// TIA Portal project "Gip & module 1" (V14)

(* hardware
DEVICE "S7-1200 station_1"  S7-1200 Station
   slot 0: "Rack_0"  S7-1200 Rack  Rack  V1.0
   slot 1: "PLC_1"  CPU 1214C DC/DC/DC  6ES7 214-1AG31-0XB0  V3.0
      slot 3: "AQ 1x12BIT_1"  AQ1 signal board  6ES7 232-4HA30-0XB0  V1.0
   slot 101: "CM 1243-5"  CM 1243-5  6GK7 243-5DX30-0XE0  V1.3
DEVICE "HMI_1"  KTP700 Basic PN
   slot 0: "KTP700 Basic PN"  KTP700 Basic PN  6AV2 123-2GB03-0AX0  14.0.1.0
   slot 1: "HMI_RT_1"  KTP700 Basic PN  6AV2 123-2GB03-0AX0  14.0.1.0
   slot 5: "HMI_1.IE_CP_1"  PROFINET Interface  14.0.1.0
      slot 1: "PROFINET Interface_1"  PROFINET Interface
         slot 1: "Port_1"  Port
DEVICE "GSD device_1"  GSD.Device
   slot 0: "Rack_0"  Rail
*)

// ===== PLC "PLC_1"  CPU 1214C DC/DC/DC =====

VAR_GLOBAL   // PLC tag table "Default tag table"
   "sensor" AT %I0.0 : Bool;
   "TBG_B_Achter" AT %I2.0 : Bool;
   "TBG_B_Midden" AT %I2.1 : Bool;
   "TBG_B_Voor" AT %I2.2 : Bool;
   "TBK_B_Achter" AT %I2.3 : Bool;
   "TBK_B_Midden" AT %I2.4 : Bool;
   "TBK_B_Voor" AT %I2.5 : Bool;
   "Brug_B_G" AT %I2.6 : Bool;
   "Brug_B_K" AT %I2.7 : Bool;
   "Brug_B_A" AT %I3.0 : Bool;
   "K1_B_Boven" AT %I3.1 : Bool;
   "K1_B_Beneden" AT %I3.2 : Bool;
   "K1_B_Vacium" AT %I3.3 : Bool;
   "Druk" AT %I3.5 : Bool;
   "TBA_B" AT %I3.4 : Bool;
   "TBG_M_Achter" AT %Q2.0 : Bool;
   "TBG_M_Voor" AT %Q2.1 : Bool;
   "TBK_M_Achter" AT %Q2.2 : Bool;
   "TBK_M_Voor" AT %Q2.3 : Bool;
   "TBA_M_Achter" AT %Q2.4 : Bool;
   "TBA_M_Voor" AT %Q2.5 : Bool;
   "Brug_M_Links" AT %Q2.6 : Bool;
   "Brug_M_Rechts" AT %Q2.7 : Bool;
   "K1_Boven" AT %Q3.0 : Bool;
   "K1_Beneden" AT %Q3.1 : Bool;
   "K1_Vacium" AT %Q3.2 : Bool;
   "Veilig opstartventiel" AT %Q3.3 : Bool;
   "New_Order" AT %M0.1 : Bool;
   "TBG_M_Achter_SR" AT %M10.0 : Bool;
   "TBG_M_Voor_SR" AT %M10.1 : Bool;
   "TBK_M_Achter_SR" AT %M10.2 : Bool;
   "TBK_M_Voor_SR" AT %M10.3 : Bool;
   "TBA_M_Achter_SR" AT %M10.4 : Bool;
   "TBA_M_Voor_SR" AT %M10.5 : Bool;
   "Brug_M_Rechts_SR" AT %M10.6 : Bool;
   "Brug_M_Links_SR" AT %M10.7 : Bool;
   "K1_Boven_SR" AT %M11.0 : Bool;
   "K1_Beneden_SR" AT %M11.1 : Bool;
   "K1_Vacium_SR" AT %M11.2 : Bool;
   "Reset_SR" AT %M11.3 : Bool;
   "S/S_SR" AT %M11.4 : Bool;
   "Start" AT %M20.0 : Bool;
   "Stop" AT %M20.1 : Bool;
   "Reset" AT %M20.2 : Bool;
   "Klein" AT %M20.3 : Bool;
   "Groot" AT %M20.4 : Bool;
   "Reset_Hmi" AT %M20.5 : Bool;
   "Test" AT %M20.6 : Bool;
   "Test_SR" AT %M11.5 : Bool;
   "Stop Alles" AT %M20.7 : Bool;
   "Proces_Order" AT %M21.0 : Bool;
END_VAR

DATA_BLOCK "Data_block_1"   // DB100
{ S7_Optimized_Access := 'FALSE' }
VERSION : 0.1
   VAR
      R : Int := 0;
      G : Int := 0;
      "B" : Int := 0;
      "G/K" : Int := 0;
      Locatie : Int;
      New : Bool := False;
   END_VAR
BEGIN
END_DATA_BLOCK

// folder: System blocks/Program resources

DATA_BLOCK "IEC_Timer_0_DB"   // DB1
{ S7_Optimized_Access := 'TRUE' }
AUTHOR : Simatic
FAMILY : IEC
NAME : IEC_TMR
VERSION : 1.0
// stored: InstanceOfName IEC_TIMER
"IEC_TIMER"
BEGIN
END_DATA_BLOCK

// folder: (top level)

FUNCTION "Block_1" : Void   // FC1, SCL
{ S7_Optimized_Access := 'TRUE' }
VERSION : 0.1
BEGIN
   IF "New_Order" = TRUE THEN
       "Data_block_1".New := TRUE;
       "New_Order" := FALSE;
   END_IF;

   IF "Data_block_1"."G/K" = 1 THEN
       "Groot" := TRUE;
       "Klein" := FALSE;
   END_IF;

   IF "Data_block_1"."G/K" = 0 THEN
       "Groot" := FALSE;
       "Klein" := TRUE;
   END_IF;
END_FUNCTION

FUNCTION "S/S + Reset + Druk" : Void   // FC2, LAD
{ S7_Optimized_Access := 'TRUE' }
VERSION : 0.1
BEGIN

REGION Network 1: S+R/S veilig opstartvetiel
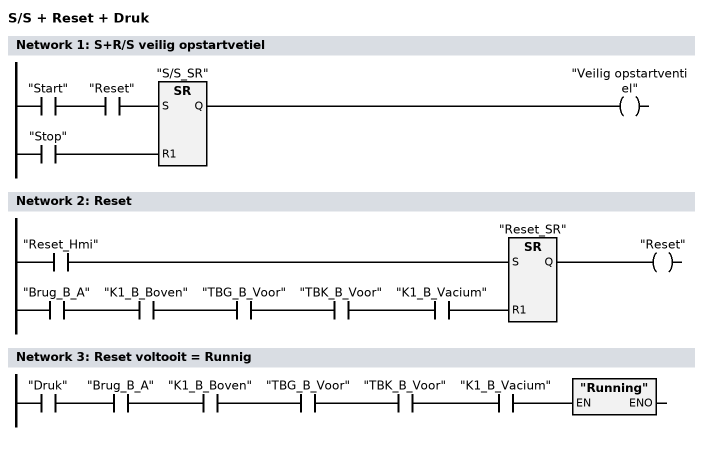
   RUNG wire#powerrail
      Contact( "Start" )
      Contact( "Reset" )
      S_SR(operand := "S/S_SR", r1 := wire#w1)
      Coil( "Veilig opstartventiel" )
   END_RUNG
   RUNG wire#powerrail
      Contact( "Stop" )
   END_RUNG wire#w1
   // the same network as SCL:
   IF "Start" AND "Reset" THEN
       "S/S_SR" := TRUE;   // SR flip-flop
   END_IF;
   IF "Stop" THEN "S/S_SR" := FALSE; END_IF;
   "Veilig opstartventiel" := "S/S_SR";
END_REGION

REGION Network 2: Reset
   RUNG wire#powerrail
      Contact( "Reset_Hmi" )
      S_SR(operand := "Reset_SR", r1 := wire#w1)
      Coil( "Reset" )
   END_RUNG
   RUNG wire#powerrail
      Contact( "Brug_B_A" )
      Contact( "K1_B_Boven" )
      Contact( "TBG_B_Voor" )
      Contact( "TBK_B_Voor" )
      Contact( "K1_B_Vacium" )
   END_RUNG wire#w1
   // the same network as SCL:
   IF "Reset_Hmi" THEN
       "Reset_SR" := TRUE;   // SR flip-flop
   END_IF;
   IF "Brug_B_A" AND "K1_B_Boven" AND "TBG_B_Voor" AND "TBK_B_Voor" AND "K1_B_Vacium" THEN
       "Reset_SR" := FALSE;
   END_IF;
   "Reset" := "Reset_SR";
END_REGION

REGION Network 3: Reset voltooit = Runnig
   RUNG wire#powerrail
      Contact( "Druk" )
      Contact( "Brug_B_A" )
      Contact( "K1_B_Boven" )
      Contact( "TBG_B_Voor" )
      Contact( "TBK_B_Voor" )
      Contact( "K1_B_Vacium" )
      "Running"()
   END_RUNG
   // the same network as SCL:
   IF "Druk" AND "Brug_B_A" AND "K1_B_Boven" AND "TBG_B_Voor" AND "TBK_B_Voor" AND "K1_B_Vacium" THEN
       "Running"();
   END_IF;
END_REGION
END_FUNCTION

FUNCTION "Running" : Void   // FC3, LAD
{ S7_Optimized_Access := 'TRUE' }
VERSION : 0.1
BEGIN

REGION Network 1: Grote bakjes naar achter
END_REGION

REGION Network 2: Grote bakjes naar voor
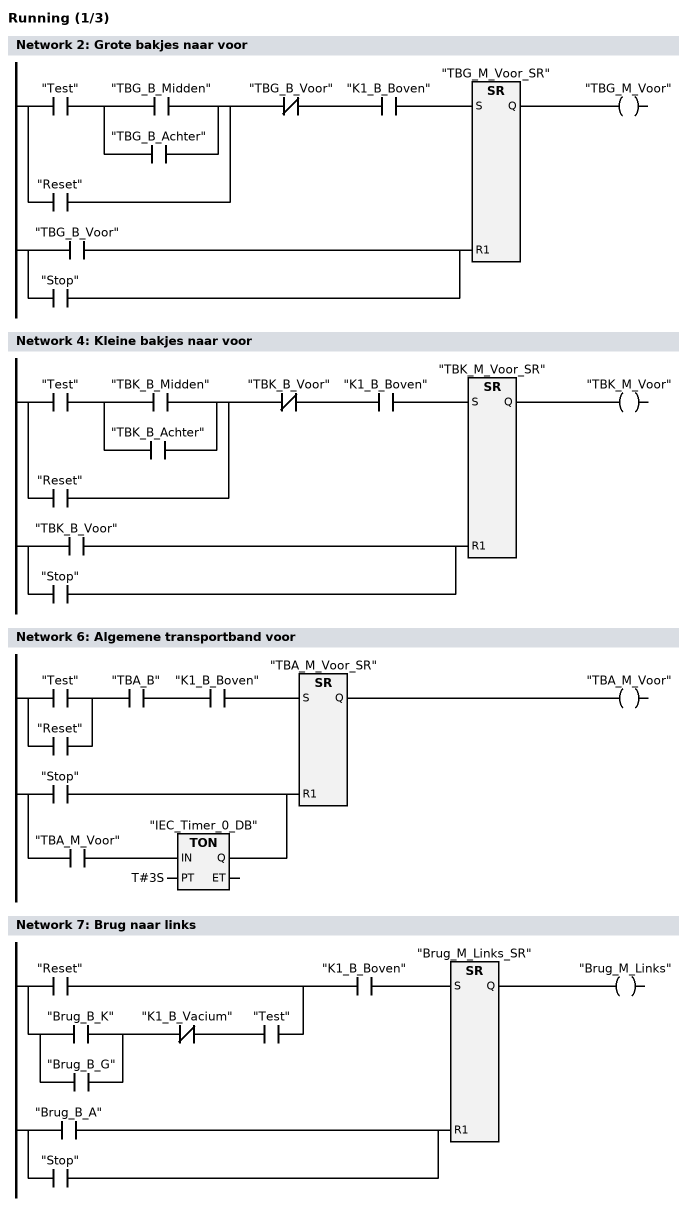
   RUNG wire#powerrail
      Contact( "Test" )
      wire#w1
      Contact( "TBG_B_Midden" )
      wire#w2
      I_Contact( "TBG_B_Voor" )
      Contact( "K1_B_Boven" )
      S_SR(operand := "TBG_M_Voor_SR", r1 := wire#w3)
      Coil( "TBG_M_Voor" )
   END_RUNG
   RUNG wire#w1
      Contact( "TBG_B_Achter" )
   END_RUNG wire#w2
   RUNG wire#powerrail
      Contact( "Reset" )
   END_RUNG wire#w2
   RUNG wire#powerrail
      Contact( "TBG_B_Voor" )
   END_RUNG wire#w3
   RUNG wire#powerrail
      Contact( "Stop" )
   END_RUNG wire#w3
   // the same network as SCL:
   IF (("Test" AND ("TBG_B_Midden" OR "TBG_B_Achter")) OR "Reset") AND NOT "TBG_B_Voor" AND "K1_B_Boven" THEN
       "TBG_M_Voor_SR" := TRUE;   // SR flip-flop
   END_IF;
   IF "TBG_B_Voor" OR "Stop" THEN "TBG_M_Voor_SR" := FALSE; END_IF;
   "TBG_M_Voor" := "TBG_M_Voor_SR";
END_REGION

REGION Network 3: Kleine bakjes naar achter
END_REGION

REGION Network 4: Kleine bakjes naar voor
   RUNG wire#powerrail
      Contact( "Test" )
      wire#w1
      Contact( "TBK_B_Midden" )
      wire#w2
      I_Contact( "TBK_B_Voor" )
      Contact( "K1_B_Boven" )
      S_SR(operand := "TBK_M_Voor_SR", r1 := wire#w3)
      Coil( "TBK_M_Voor" )
   END_RUNG
   RUNG wire#w1
      Contact( "TBK_B_Achter" )
   END_RUNG wire#w2
   RUNG wire#powerrail
      Contact( "Reset" )
   END_RUNG wire#w2
   RUNG wire#powerrail
      Contact( "TBK_B_Voor" )
   END_RUNG wire#w3
   RUNG wire#powerrail
      Contact( "Stop" )
   END_RUNG wire#w3
   // the same network as SCL:
   IF (("Test" AND ("TBK_B_Midden" OR "TBK_B_Achter")) OR "Reset") AND NOT "TBK_B_Voor" AND "K1_B_Boven" THEN
       "TBK_M_Voor_SR" := TRUE;   // SR flip-flop
   END_IF;
   IF "TBK_B_Voor" OR "Stop" THEN "TBK_M_Voor_SR" := FALSE; END_IF;
   "TBK_M_Voor" := "TBK_M_Voor_SR";
END_REGION

REGION Network 5: Algemene transportband achter
END_REGION

REGION Network 6: Algemene transportband voor
   "IEC_Timer_0_DB".TON(IN := "TBA_M_Voor", PT := T#3S);
   IF ("Test" OR "Reset") AND "TBA_B" AND "K1_B_Boven" THEN
       "TBA_M_Voor_SR" := TRUE;   // SR flip-flop
   END_IF;
   IF "Stop" OR "IEC_Timer_0_DB".Q THEN "TBA_M_Voor_SR" := FALSE; END_IF;
   "TBA_M_Voor" := "TBA_M_Voor_SR";
END_REGION

REGION Network 7: Brug naar links
   RUNG wire#powerrail
      Contact( "Reset" )
      wire#w1
      Contact( "K1_B_Boven" )
      S_SR(operand := "Brug_M_Links_SR", r1 := wire#w3)
      Coil( "Brug_M_Links" )
   END_RUNG
   RUNG wire#powerrail
      Contact( "Brug_B_K" )
      wire#w2
      I_Contact( "K1_B_Vacium" )
      Contact( "Test" )
   END_RUNG wire#w1
   RUNG wire#powerrail
      Contact( "Brug_B_G" )
   END_RUNG wire#w2
   RUNG wire#powerrail
      Contact( "Brug_B_A" )
   END_RUNG wire#w3
   RUNG wire#powerrail
      Contact( "Stop" )
   END_RUNG wire#w3
   // the same network as SCL:
   IF ("Reset" OR (("Brug_B_K" OR "Brug_B_G") AND NOT "K1_B_Vacium" AND "Test")) AND "K1_B_Boven" THEN
       "Brug_M_Links_SR" := TRUE;   // SR flip-flop
   END_IF;
   IF "Brug_B_A" OR "Stop" THEN "Brug_M_Links_SR" := FALSE; END_IF;
   "Brug_M_Links" := "Brug_M_Links_SR";
END_REGION

REGION Network 8: Brug naar rechts
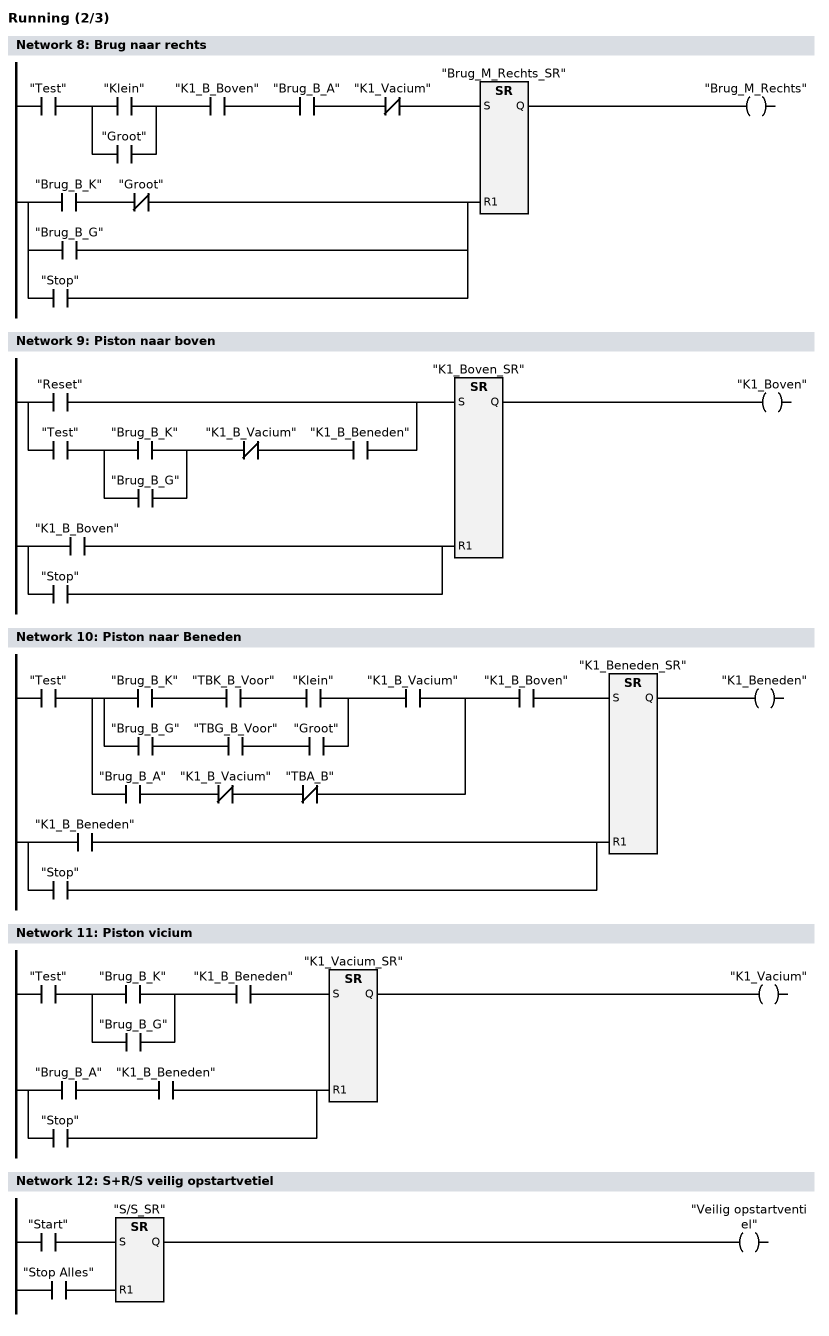
   RUNG wire#powerrail
      Contact( "Test" )
      wire#w1
      Contact( "Klein" )
      wire#w2
      Contact( "K1_B_Boven" )
      Contact( "Brug_B_A" )
      I_Contact( "K1_Vacium" )
      S_SR(operand := "Brug_M_Rechts_SR", r1 := wire#w3)
      Coil( "Brug_M_Rechts" )
   END_RUNG
   RUNG wire#w1
      Contact( "Groot" )
   END_RUNG wire#w2
   RUNG wire#powerrail
      Contact( "Brug_B_K" )
      I_Contact( "Groot" )
   END_RUNG wire#w3
   RUNG wire#powerrail
      Contact( "Brug_B_G" )
   END_RUNG wire#w3
   RUNG wire#powerrail
      Contact( "Stop" )
   END_RUNG wire#w3
   // the same network as SCL:
   IF "Test" AND ("Klein" OR "Groot") AND "K1_B_Boven" AND "Brug_B_A" AND NOT "K1_Vacium" THEN
       "Brug_M_Rechts_SR" := TRUE;   // SR flip-flop
   END_IF;
   IF ("Brug_B_K" AND NOT "Groot") OR "Brug_B_G" OR "Stop" THEN "Brug_M_Rechts_SR" := FALSE; END_IF;
   "Brug_M_Rechts" := "Brug_M_Rechts_SR";
END_REGION

REGION Network 9: Piston naar boven
   RUNG wire#powerrail
      Contact( "Reset" )
      wire#w1
      S_SR(operand := "K1_Boven_SR", r1 := wire#w4)
      Coil( "K1_Boven" )
   END_RUNG
   RUNG wire#powerrail
      Contact( "Test" )
      wire#w2
      Contact( "Brug_B_K" )
      wire#w3
      I_Contact( "K1_B_Vacium" )
      Contact( "K1_B_Beneden" )
   END_RUNG wire#w1
   RUNG wire#w2
      Contact( "Brug_B_G" )
   END_RUNG wire#w3
   RUNG wire#powerrail
      Contact( "K1_B_Boven" )
   END_RUNG wire#w4
   RUNG wire#powerrail
      Contact( "Stop" )
   END_RUNG wire#w4
   // the same network as SCL:
   IF "Reset" OR ("Test" AND ("Brug_B_K" OR "Brug_B_G") AND NOT "K1_B_Vacium" AND "K1_B_Beneden") THEN
       "K1_Boven_SR" := TRUE;   // SR flip-flop
   END_IF;
   IF "K1_B_Boven" OR "Stop" THEN "K1_Boven_SR" := FALSE; END_IF;
   "K1_Boven" := "K1_Boven_SR";
END_REGION

REGION Network 10: Piston naar Beneden
   RUNG wire#powerrail
      Contact( "Test" )
      wire#w1
      Contact( "Brug_B_K" )
      Contact( "TBK_B_Voor" )
      Contact( "Klein" )
      wire#w2
      Contact( "K1_B_Vacium" )
      wire#w3
      Contact( "K1_B_Boven" )
      S_SR(operand := "K1_Beneden_SR", r1 := wire#w4)
      Coil( "K1_Beneden" )
   END_RUNG
   RUNG wire#w1
      Contact( "Brug_B_G" )
      Contact( "TBG_B_Voor" )
      Contact( "Groot" )
   END_RUNG wire#w2
   RUNG wire#w1
      Contact( "Brug_B_A" )
      I_Contact( "K1_B_Vacium" )
      I_Contact( "TBA_B" )
   END_RUNG wire#w3
   RUNG wire#powerrail
      Contact( "K1_B_Beneden" )
   END_RUNG wire#w4
   RUNG wire#powerrail
      Contact( "Stop" )
   END_RUNG wire#w4
   // the same network as SCL:
   IF "Test" AND (((("Brug_B_K" AND "TBK_B_Voor" AND "Klein") OR ("Brug_B_G" AND "TBG_B_Voor" AND "Groot")) AND "K1_B_Vacium") OR ("Brug_B_A" AND NOT "K1_B_Vacium" AND NOT "TBA_B")) AND "K1_B_Boven" THEN
       "K1_Beneden_SR" := TRUE;   // SR flip-flop
   END_IF;
   IF "K1_B_Beneden" OR "Stop" THEN "K1_Beneden_SR" := FALSE; END_IF;
   "K1_Beneden" := "K1_Beneden_SR";
END_REGION

REGION Network 11: Piston vicium
   RUNG wire#powerrail
      Contact( "Test" )
      wire#w1
      Contact( "Brug_B_K" )
      wire#w2
      Contact( "K1_B_Beneden" )
      S_SR(operand := "K1_Vacium_SR", r1 := wire#w3)
      Coil( "K1_Vacium" )
   END_RUNG
   RUNG wire#w1
      Contact( "Brug_B_G" )
   END_RUNG wire#w2
   RUNG wire#powerrail
      Contact( "Brug_B_A" )
      Contact( "K1_B_Beneden" )
   END_RUNG wire#w3
   RUNG wire#powerrail
      Contact( "Stop" )
   END_RUNG wire#w3
   // the same network as SCL:
   IF "Test" AND ("Brug_B_K" OR "Brug_B_G") AND "K1_B_Beneden" THEN
       "K1_Vacium_SR" := TRUE;   // SR flip-flop
   END_IF;
   IF ("Brug_B_A" AND "K1_B_Beneden") OR "Stop" THEN "K1_Vacium_SR" := FALSE; END_IF;
   "K1_Vacium" := "K1_Vacium_SR";
END_REGION

REGION Network 12: S+R/S veilig opstartvetiel
   RUNG wire#powerrail
      Contact( "Start" )
      S_SR(operand := "S/S_SR", r1 := wire#w1)
      Coil( "Veilig opstartventiel" )
   END_RUNG
   RUNG wire#powerrail
      Contact( "Stop Alles" )
   END_RUNG wire#w1
   // the same network as SCL:
   IF "Start" THEN
       "S/S_SR" := TRUE;   // SR flip-flop
   END_IF;
   IF "Stop Alles" THEN "S/S_SR" := FALSE; END_IF;
   "Veilig opstartventiel" := "S/S_SR";
END_REGION

REGION Network 13: Reset
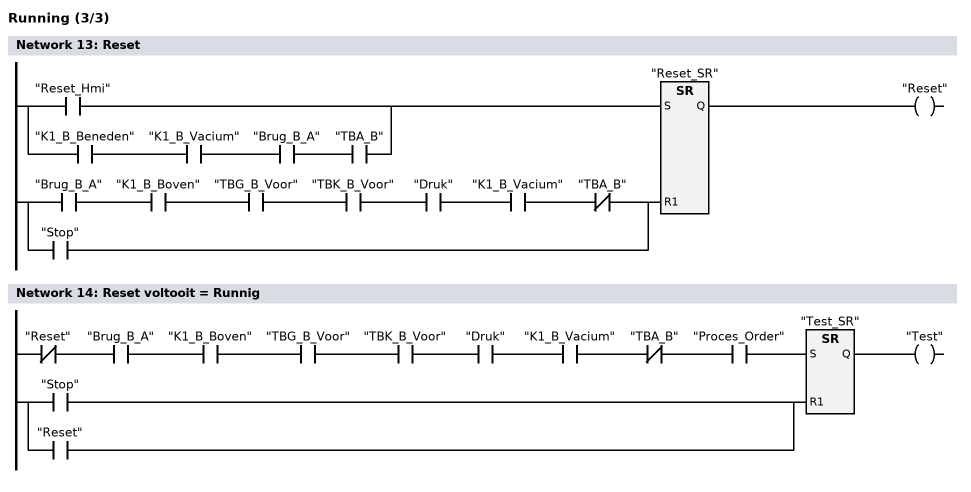
   RUNG wire#powerrail
      Contact( "Reset_Hmi" )
      wire#w1
      S_SR(operand := "Reset_SR", r1 := wire#w2)
      Coil( "Reset" )
   END_RUNG
   RUNG wire#powerrail
      Contact( "K1_B_Beneden" )
      Contact( "K1_B_Vacium" )
      Contact( "Brug_B_A" )
      Contact( "TBA_B" )
   END_RUNG wire#w1
   RUNG wire#powerrail
      Contact( "Brug_B_A" )
      Contact( "K1_B_Boven" )
      Contact( "TBG_B_Voor" )
      Contact( "TBK_B_Voor" )
      Contact( "Druk" )
      Contact( "K1_B_Vacium" )
      I_Contact( "TBA_B" )
   END_RUNG wire#w2
   RUNG wire#powerrail
      Contact( "Stop" )
   END_RUNG wire#w2
   // the same network as SCL:
   IF "Reset_Hmi" OR ("K1_B_Beneden" AND "K1_B_Vacium" AND "Brug_B_A" AND "TBA_B") THEN
       "Reset_SR" := TRUE;   // SR flip-flop
   END_IF;
   IF ("Brug_B_A" AND "K1_B_Boven" AND "TBG_B_Voor" AND "TBK_B_Voor" AND "Druk" AND "K1_B_Vacium" AND NOT "TBA_B") OR "Stop" THEN
       "Reset_SR" := FALSE;
   END_IF;
   "Reset" := "Reset_SR";
END_REGION

REGION Network 14: Reset voltooit = Runnig
   RUNG wire#powerrail
      I_Contact( "Reset" )
      Contact( "Brug_B_A" )
      Contact( "K1_B_Boven" )
      Contact( "TBG_B_Voor" )
      Contact( "TBK_B_Voor" )
      Contact( "Druk" )
      Contact( "K1_B_Vacium" )
      I_Contact( "TBA_B" )
      Contact( "Proces_Order" )
      S_SR(operand := "Test_SR", r1 := wire#w1)
      Coil( "Test" )
   END_RUNG
   RUNG wire#powerrail
      Contact( "Stop" )
   END_RUNG wire#w1
   RUNG wire#powerrail
      Contact( "Reset" )
   END_RUNG wire#w1
   // the same network as SCL:
   IF NOT "Reset" AND "Brug_B_A" AND "K1_B_Boven" AND "TBG_B_Voor" AND "TBK_B_Voor" AND "Druk" AND "K1_B_Vacium" AND NOT "TBA_B" AND "Proces_Order" THEN
       "Test_SR" := TRUE;   // SR flip-flop
   END_IF;
   IF "Stop" OR "Reset" THEN "Test_SR" := FALSE; END_IF;
   "Test" := "Test_SR";
END_REGION
END_FUNCTION

ORGANIZATION_BLOCK "Main"   // OB1, LAD, ProgramCycle
TITLE = "Main Program Sweep (Cycle)"
{ S7_Optimized_Access := 'TRUE' }
VERSION : 0.1
   VAR_TEMP
      sensor_Memorie : Bool;
   END_VAR
BEGIN

REGION Network 1
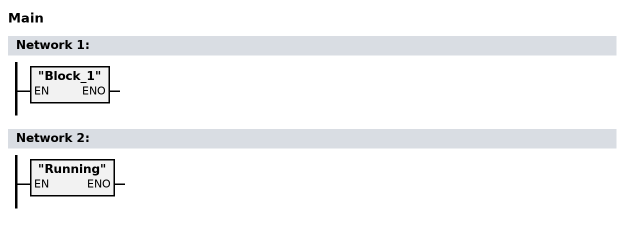
   RUNG wire#powerrail
      "Block_1"()
   END_RUNG
   // the same network as SCL:
   "Block_1"();
END_REGION

REGION Network 2
   RUNG wire#powerrail
      "Running"()
   END_RUNG
   // the same network as SCL:
   "Running"();
END_REGION
END_ORGANIZATION_BLOCK

(* ===== HMI "HMI_RT_1" =====
system functions are stored by id; their names below are inferred from use
connection "HMI_Connection_1": ETHERNET, SMART_S7_1200_OMS

HMI tags "Default tag table"
   "Tag_ScreenNumber" : UInt, internal
   "sensor" : Bool = PLC sensor AT %I0.0, 1 s
   "Data_block_1_R" : Int = PLC Data_block_1.R AT %DB100.DBW0, 1 s
   "Data_block_1_B" : Int = PLC Data_block_1.B AT %DB100.DBW4, 1 s
   "Data_block_1_G" : Int = PLC Data_block_1.G AT %DB100.DBW2, 1 s
   "Data_block_1_G/K" : Int = PLC Data_block_1.G/K AT %DB100.DBW6, 1 s
   "Data_block_1_Locatie" : Int = PLC Data_block_1.Locatie AT %DB100.DBW8, 1 s
   "New_Order" : Bool = PLC New_Order AT %M0.1, 1 s
   "Start" : Bool = PLC Start AT %M20.0, 1 s
   "Stop" : Bool = PLC Stop AT %M20.1, 1 s
   "Reset_Hmi" : Bool = PLC Reset_Hmi AT %M20.5, 1 s
   "Stop Alles" : Bool = PLC "Stop Alles" AT %M20.7, 1 s
   "Proces_Order" : Bool = PLC Proces_Order AT %M21.0, 1 s

screen "Root screen" 800x480, template "Template_1"
   on GenerateScreen: SetTag("Tag_ScreenNumber", 1)
   TextField "Text field_1" at 13,62 size 64x28; Text 'Rood:'
   TextField "Text field_2" at 13,106 size 73x28; Text 'Groen:'
   TextField "Text field_3" at 13,150 size 75x28; Text 'Blauw:'
   TextField "Text field_4" at 13,238 size 84x28; Text 'Locatie:'
   TextField "Text field_5" at 13,194 size 53x28; Text 'G/K:'
   IOField "I/O field_1" at 104,62 size 24x32; FormatPattern 9
      ProcessValue <- "Data_block_1_R"
   IOField "I/O field_2" at 104,106 size 24x32; FormatPattern 9
      ProcessValue <- "Data_block_1_G"
   IOField "I/O field_3" at 104,150 size 24x32; FormatPattern 9
      ProcessValue <- "Data_block_1_B"
   IOField "I/O field_4" at 104,194 size 24x32; FormatPattern 9
      ProcessValue <- "Data_block_1_G/K"
   IOField "I/O field_5" at 104,238 size 24x32; FormatPattern 9
      ProcessValue <- "Data_block_1_Locatie"
   Button "Button_1" at 13,290 size 113x42; TextOff 'New Order'
      on Press: SetBit("New_Order")
   Button "Button_2" at 172,290 size 113x42; TextOff 'Start'
      on Press: SetBit("Start")
      on Release: ResetBit("Start")
   Button "Button_3" at 331,290 size 113x42; TextOff 'Stop'
      on Press: SetBit("Stop")
      on Release: ResetBit("Stop")
   Button "Button_4" at 490,290 size 113x42; TextOff 'Reset'
      on Press: SetBit("Reset_Hmi")
      on Release: ResetBit("Reset_Hmi")
   Button "Button_5" at 331,349 size 113x42; TextOff 'Stop Druk'
      on Release: ResetBit("Stop Alles")
      on Press: SetBit("Stop Alles")
   Button "Button_6" at 13,349 size 113x42; TextOff 'Start Order'
      on Press: SetBit("Proces_Order")
      on Release: ResetBit("Proces_Order")

Template "Template_1" 800x480
   Button "Exit" at 714,429 size 71x50; TextOn 'Exit'; TextOff 'Exit'; PictureOn "ExitRuntime_KTP700_Basic_PN_TR"; PictureOff "ExitRuntime_KTP700_Basic_PN_TR"
      on Release: StopRuntime(0)
   Button "Template_Button" at 614,429 size 71x50; TextOff 'Text'
   Button "Template_Button_1" at 514,429 size 71x50; TextOff 'Text'
   Button "Template_Button_2" at 414,429 size 71x50; TextOff 'Text'
   Button "Template_Button_3" at 314,429 size 71x50; TextOff 'Text'
   Button "Template_Button_4" at 214,429 size 71x50; TextOff 'Text'
   Button "Template_Button_5" at 114,429 size 71x50; TextOff 'Text'
   Button "Start screen" at 14,429 size 71x50; TextOn 'Start screen'; TextOff 'Start screen'; PictureOn "NavigateHome_KTP700_Basic_PN_TR"; PictureOff "NavigateHome_KTP700_Basic_PN_TR"
      on Release: ActivateScreen("Root screen", 0)
   SymbolicIOField "Symbolic_IO_Field_Screen" at 93,9 size 600x33; TextOn '1'; TextOff '0'; TextList "TextList_ScreenNames"
      on Change: ActivateScreenByNumber("Tag_ScreenNumber", 0)
      ProcessValue <- "Tag_ScreenNumber"
   DateTimeField "HmiScreenItemData" at 695,25 size 105x25
   DateTimeField "HmiScreenItemData_1" at 695,0 size 105x25
   GraphicView "Logo" at 0,0 size 91x51; Picture "Logo of HMI_1"
*)